// Mitsubishi GX Works2 project: 11-06-2020 Counter   PLC: FX3G

PROGRAM MAIN
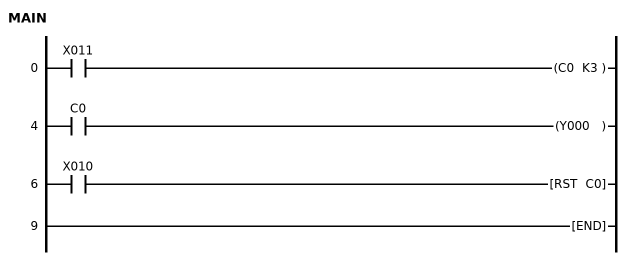
0     LD      X011
      OUT     C0 K3
4     LD      C0
      OUT     Y000
6     LD      X010
      RST     C0
9     END
END_PROGRAM
